{attribute 'GeneratedUsingTerminal: EL9570--0000'}
{attribute addProperty BoxType "EL9570--0000"}
{attribute addProperty Description "EL9570 Buffer capacitor terminal"}
{attribute addProperty Physics "KK"}
{attribute addProperty Id "EL9570"}
{attribute addProperty CRC "837845432"}
{attribute addProperty Size "0"}
TYPE EL9570_31F081B8 EXTENDS EtcSlaveTerminalBase_947E5A46 :
STRUCT
END_STRUCT
END_TYPE

(* stored: Version 1.2.0.0, ProductVersion 3.1.4024.9
   DUT EL9570_31F081B8: Id {b12f7142-be49-43c0-a22b-4c8dbf872ec3} *)
